// TIA Portal V19 export
TYPE "UDT_TANKPRESS_2"
   STRUCT
      r { S7_SetPoint := 'True'} : Real;
      d { S7_SetPoint := 'True'} : Real;
      hPt { S7_SetPoint := 'True'} : Real;
      hBase { S7_SetPoint := 'True'} : Real;
      hCyl { S7_SetPoint := 'True'} : Real;
      hAct : Real;
      vol : Real;
   END_STRUCT;
END_TYPE
